// TwinCAT 3 PLC project Main_PLC
// ProgramVersion: 3.1.4024.0
// libraries:
//   Tc2_Math, * (Beckhoff Automation GmbH)
//   Tc2_Standard, * (Beckhoff Automation GmbH)
//   Tc2_System, * (Beckhoff Automation GmbH)
//   Tc3_Module, * (Beckhoff Automation GmbH)
// project tree:
//   DUTs/ E_Mode.TcDUT, ST_HmiControl.TcDUT, ST_AutoControlSwitch.TcDUT
//   GVLs/ gHMI.TcGVL, gIO.TcGVL
//   / PlcTask.TcTTO
//   POUs/Function Blocks/ FB_MockTank.TcPOU, FB_StopWatch.TcPOU, FB_SwitchSingleThrow.TcPOU, FB_TankControl.TcPOU
//   POUs/Function/Utilities/ F_Clear.TcPOU, F_Compare.TcPOU, F_Copy.TcPOU
//   POUs/ MAIN.TcPOU
// real-time tasks:
//   TASK PlcTask: cycle T#10ms, priority 20, ADS port 350
// I/O:
//   DEVICE EtherCAT Interface 1 (EK1100) (disabled), AmsNetId 10.186.0.125.2.1
//     Coupler 1 [EK1100 EtherCAT Coupler (2A E-Bus)]
//       Digital Input 1 (EL1008) [EL1008 8Ch. Dig. Input 24V, 3ms]
//       Digital Output 1 (EL2008) [EL2008 8Ch. Dig. Output 24V, 0.5A]
// variable links:
//   Main PLC/Main PLC Instance <-> EtherCAT Interface 1 (EK1100)/Coupler 1/Digital Input 1 (EL1008)
//     PlcTask Inputs/gIO.I[{0..7}] <-> Channel {1..8}/Input  (8 links)
//   Main PLC/Main PLC Instance <-> EtherCAT Interface 1 (EK1100)/Coupler 1/Digital Output 1 (EL2008)
//     PlcTask Outputs/gIO.Q[{0..7}] <-> Channel {1..8}/Output  (8 links)

CONFIGURATION Main_PLC
    RESOURCE PLC ON TwinCAT3
        TASK PlcTask(INTERVAL := T#10ms, PRIORITY := 20);
        PROGRAM MAIN WITH PlcTask : MAIN;
    END_RESOURCE
END_CONFIGURATION

// ---- DUTs/E_Mode.TcDUT
{attribute 'qualified_only'}
{attribute 'strict'}
TYPE E_Mode :
(
	Manual, Auto
)USINT;
END_TYPE

// ---- DUTs/ST_HmiControl.TcDUT
TYPE ST_HmiControl :
STRUCT
	Lamp: WORD;
	Button: WORD;
	Interlock: WORD;
END_STRUCT
END_TYPE

// ---- DUTs/ST_AutoControlSwitch.TcDUT
TYPE ST_AutoControlSwitch :
STRUCT
	bExecute: BOOL;
	bDone: BOOL;
	bError: BOOL;
END_STRUCT
END_TYPE

// ---- GVLs/gHMI.TcGVL
{attribute 'qualified_only'}
VAR_GLOBAL
END_VAR

// ---- GVLs/gIO.TcGVL
VAR_GLOBAL
	I AT %I*: ARRAY[0..7] OF BOOL;
	Q AT %Q*: ARRAY[0..7] OF BOOL;
END_VAR

// ---- POUs/MAIN.TcPOU
PROGRAM MAIN
VAR
	fbTankControl: FB_TankControl;
	fbMockTank: FB_MockTank;
	
	{attribute 'OPC.UA.DA' := '1'}
	stTankPumpCtrl: ST_HmiControl;
	
	{attribute 'OPC.UA.DA' := '1'}
	bHmiReset: BOOL;
	
	{attribute 'OPC.UA.DA' := '1'}
	eHmiMode: E_Mode;
	
	{attribute 'OPC.UA.DA':='1'}
	{attribute 'OPC.UA.DA.Access':='1'}
	rTankVolume: REAL;
	
	{attribute 'OPC.UA.DA':='1'}
	{attribute 'OPC.UA.DA.Access':='1'}
	rConsumptionRate: REAL;
	
	{attribute 'OPC.UA.DA':='1'}
	{attribute 'OPC.UA.DA.Access':='1'}
	nAlarmBits: DWORD;
	
	nLiveAlarmBits: DWORD;
END_VAR

fbMockTank(
	bEnable:= fbMockTank.bEnable, 
	bPumpOn:= Q[0], 
	rPumpFillRate:= fbMockTank.rPumpFillRate, 
	rCapacity:= fbMockTank.rCapacity, 
	tSamplingRate:= fbMockTank.tSamplingRate,
	nLowLevelSensorPos:= fbMockTank.nLowLevelSensorPos, 
	nHighLevelSensorPos:= fbMockTank.nHighLevelSensorPos, 
	rVolume=> rTankVolume, 
	rConsumption=> rConsumptionRate, 
	bLowLevel=>, 
	bHighLevel=> );

IF fbMockTank.bEnable THEN	
	I[0]:= fbMockTank.bLowLevel;
	I[1]:= fbMockTank.bHighLevel;
END_IF

fbTankControl(
	bEnableFillTimeout:= fbTankControl.bEnableFillTimeout, 
	eMode:= eHmiMode, 
	bReset:= fbTankControl.bReset, 
	tHighLevelSensorDly:= fbTankControl.tHighLevelSensorDly, 
	tLowLevelSensorDly:= fbTankControl.tLowLevelSensorDly, 
	tFillTimeout:= fbTankControl.tFillTimeout, 
	bPumpOnOutput:= Q[0], 
	bHighLevelSensor:= I[1], 
	bLowLevelSensor:= I[0], 
	stPumpHmiControl:= stTankPumpCtrl);
	
IF bHmiReset THEN
	F_Clear(nAlarmBits);
END_IF

nLiveAlarmBits.0:= NOT I[0];
nLiveAlarmBits.1:= I[1];

nAlarmBits:= nAlarmBits OR nLiveAlarmBits;

END_PROGRAM

// ---- POUs/Function Blocks/FB_TankControl.TcPOU
FUNCTION_BLOCK FB_TankControl
VAR_INPUT
	bEnableFillTimeout: BOOL;
	eMode: E_Mode;
	bReset: BOOL;
	tHighLevelSensorDly: TIME:= T#0.2S;
	tLowLevelSensorDly: TIME:= T#0.2S;
	tFillTimeout: TIME:= T#10S;
END_VAR
VAR_IN_OUT
	bPumpOnOutput: BOOL;
	bHighLevelSensor: BOOL;
	bLowLevelSensor: BOOL;
	stPumpHmiControl: ST_HmiControl;
END_VAR
VAR
	tonHighLevelSensorDly: TON;
	tonLowLevelSensorDly: TON;
	tonFillTimeout: TON;
	
	stPumpOnAuto: ST_AutoControlSwitch;
	fbPumpControl: FB_SwitchSingleThrow;
END_VAR

tonHighLevelSensorDly(IN:= bHighLevelSensor, PT:= tHighLevelSensorDly, Q=> , ET=> );
tonLowLevelSensorDly(IN:= NOT bLowLevelSensor, PT:= tLowLevelSensorDly, Q=> , ET=> );

tonFillTimeout(IN:= bEnableFillTimeout, PT:= tFillTimeout, Q=> , ET=> );

fbPumpControl(
	bManualMode:= eMode = E_Mode.Manual, 
	bReset:= bReset,  
	bSensor:= TRUE, 
	bInterlock:= tonHighLevelSensorDly.Q, 
	tTimeout:= , 
	tMinSensorOn:= , 
	stAuto:= stPumpOnAuto, 
	stHmiControl:= stPumpHmiControl,
	bError=> , 
	sErrorMsg=> , 
	bSwitch=> bPumpOnOutput, 
	bOverrideState=> );

IF eMode = E_Mode.Auto THEN
	stPumpOnAuto.bExecute:= 
		NOT (tonHighLevelSensorDly.Q OR tonFillTimeout.Q) AND (stPumpOnAuto.bExecute OR tonLowLevelSensorDly.Q);
END_IF

END_FUNCTION_BLOCK

// ---- POUs/Function Blocks/FB_SwitchSingleThrow.TcPOU
FUNCTION_BLOCK FB_SwitchSingleThrow
VAR_INPUT
	bManualMode: BOOL;
	bReset: BOOL;
	bSensor: BOOL;
	bInterlock: BOOL;
	tTimeout: TIME:= tDefaultTimeOut;
	tMinSensorOn: TIME:= tDefaultMinSensorOn;
END_VAR
VAR_IN_OUT
	stAuto: ST_AutoControlSwitch;
	stHmiControl: ST_HmiControl;
END_VAR
VAR_OUTPUT
	bError: BOOL;
	sErrorMsg: STRING(100);
	bSwitch: BOOL;
	
	bOverrideState: BOOL;
END_VAR
VAR
	tonPulse_Delay: Ton;
	tonSeqDelay: Ton;
	tonSeqTimeout: Ton;	
	
	rtReset: R_TRIG;
	
	nCurrentState: BYTE;
	nAutoState: BYTE;
	
	rtHome_Execute_HMI: R_TRIG;
	rtAction_Execute_HMI: R_TRIG;
	
	ton_DoneResetTimeout: TON;
	
	_bSwitch: BOOL;
END_VAR
VAR CONSTANT
	tDefaultMinPulseOn: TIME:= T#2S;
	tDefaultMinSensorOn: TIME:= T#0.1S;
	tDefaultTimeOut: TIME:= T#10S;
	tDefaultResetDone: TIME:= T#1S;
END_VAR

tonSeqDelay(
	IN:= bSensor,
	PT:= tMinSensorOn);
	
tonSeqTimeout(
	IN:= stAuto.bExecute AND NOT (stAuto.bDone OR stAuto.bError OR bManualMode),
	PT:= tTimeout);
	
ton_DoneResetTimeout(
	IN:= stAuto.bDone AND NOT bSensor,
	PT:= tDefaultResetDone);
	
IF ton_DoneResetTimeout.Q THEN
	F_Clear(stAuto.bDone);
END_IF
	
rtReset(CLK:= bReset);

bError:= stAuto.bError;

rtHome_Execute_HMI(CLK:= stHmiControl.Button.0);
rtAction_Execute_HMI(CLK:= stHmiControl.Button.1);

IF rtReset.Q AND bError THEN	
	stAuto.bError:= FALSE;
	sErrorMsg:= '';
END_IF

IF tonPulse_Delay.Q THEN
	F_Clear(stHmiControl);
	F_Clear(stAuto.bExecute);
	F_Clear(_bSwitch);
END_IF
IF bManualMode THEN
	IF rtHome_Execute_HMI.Q THEN
		stHmiControl.Button.1:= FALSE;
		_bSwitch:= FALSE;
	ELSIF rtAction_Execute_HMI.Q THEN
		IF bInterlock THEN
			stHmiControl.Button.1:= FALSE;
		ELSE
			stHmiControl.Button.0:= FALSE;
			_bSwitch:= TRUE;
		END_IF
	END_IF
	stAuto.bExecute:= stHmiControl.Button.1;
ELSE 
	IF NOT (bError AND stAuto.bExecute) THEN
		IF stAuto.bExecute THEN
			IF NOT bInterlock THEN
				_bSwitch:= TRUE;
			END_IF
		ELSE
			_bSwitch:= FALSE;
		END_IF
		IF tonSeqTimeout.Q THEN
			stAuto.bError:= TRUE;
			IF bInterlock THEN
				sErrorMsg:= 'Interlock Error';
			ELSE 
				sErrorMsg:= 'Timeout Error';
			END_IF
		END_IF
	END_IF
	stHmiControl.Button.1:= stAuto.bExecute;
	stHmiControl.Button.0:= NOT stAuto.bExecute;
END_IF

stHmiControl.Interlock.1:= bInterlock;
stAuto.bDone:= stAuto.bExecute AND (tonSeqDelay.Q OR stAuto.bDone) AND NOT stAuto.bError;

nCurrentState.0:= bSwitch;
IF NOT bManualMode THEN
	nAutoState:= nCurrentState;
END_IF
bOverrideState:= nCurrentState <> nAutoState;

bSwitch:= _bSwitch;

END_FUNCTION_BLOCK

// ---- POUs/Function/Utilities/F_Clear.TcPOU
FUNCTION F_Clear : BOOL //size of data type should not exceed double integer maximum value
VAR_INPUT
	Target: ANY;
END_VAR
VAR
END_VAR

MemSet(
	DestAddr       	:= Target.pValue, 
    FillByte    	:= 0, 
    n   			:= DINT_TO_UDINT(Target.diSize)
);

END_FUNCTION

// ---- POUs/Function Blocks/FB_MockTank.TcPOU
FUNCTION_BLOCK FB_MockTank
VAR_INPUT
	bEnable: BOOL;
	bPumpOn: BOOL;
	rPumpFillRate: REAL:= 50; //litres per second
	rCapacity: REAL:= 500; //litres
	nLowLevelSensorPos: REAL:= 0.2*rCapacity; //percent
	nHighLevelSensorPos: REAL:= 0.8*rCapacity; //percent
	tSamplingRate: TIME:= T#100MS;
END_VAR
VAR_OUTPUT
	rVolume: REAL;
	rConsumption: REAL;
	bLowLevel: BOOL;
	bHighLevel: BOOL;
END_VAR
VAR
	tonConsumptionPeriod: TON;
	rFillRate: REAL;
	fbRandom: DRAND;
	tonSamplingRate: TON;
	rFillRateFactor: REAL;
END_VAR

VAR CONSTANT
	
END_VAR

bLowLevel:= rVolume > nLowLevelSensorPos;
bHighLevel:= rVolume > nHighLevelSensorPos;

tonConsumptionPeriod(IN:= bEnable AND NOT tonConsumptionPeriod.Q, PT:= , Q=> , ET=> );
tonSamplingRate(IN:= bEnable AND NOT tonSamplingRate.Q, PT:= tSamplingRate, Q=> , ET=> );
IF bPumpOn THEN
	rFillRate:= rPumpFillRate;
ELSE
	rFillRate:= 0.0;
END_IF

IF bEnable THEN
	rFillRateFactor:= TIME_TO_REAL(tonSamplingRate.PT)/1000;
	IF tonConsumptionPeriod.Q THEN
		fbRandom(seed:=LREAL_TO_INT(fbRandom.Num));
		IF rConsumption = 0.0 THEN
			rConsumption:= fbRandom.Num*fbRandom.Num*20;
			tonConsumptionPeriod.PT:= LREAL_TO_TIME(fbRandom.Num*10000);
		ELSE
			rConsumption:= 0.0;
			tonConsumptionPeriod.PT:= LREAL_TO_TIME(fbRandom.Num*2000);
		END_IF
	END_IF
	IF rVolume < 0.1 THEN
		rConsumption:= 0.0;
	END_IF
	IF tonSamplingRate.Q THEN
		rVolume:= rVolume + (rFillRate - rConsumption)*rFillRateFactor;
	END_IF
END_IF

END_FUNCTION_BLOCK

// ---- POUs/Function Blocks/FB_StopWatch.TcPOU
FUNCTION_BLOCK FB_StopWatch
VAR_INPUT
	bStart: BOOL;
	bReset: BOOL;
END_VAR
VAR_IN_OUT
	tElapsedTime: TIME;
END_VAR
VAR
	tStartTime: TIME;
	rtReset: R_TRIG;
	tLastElapsedTime: TIME;
END_VAR

rtReset(CLK:= bReset);
IF rtReset.Q THEN
	F_Clear(tLastElapsedTime);
	F_Clear(tStartTime);
END_IF

IF bStart AND tStartTime = T#0MS THEN
	tStartTime:= TIME();
ELSIF NOT bStart AND tStartTime > T#0MS THEN
	tLastElapsedTime:= tLastElapsedTime + TIME() - tStartTime;
	F_Clear(tStartTime);
END_IF

IF tStartTime > T#0MS THEN
	tElapsedTime:= tLastElapsedTime + TIME() - tStartTime;
ELSIF tLastElapsedTime = T#0S AND tElapsedTime > T#0S THEN
	tLastElapsedTime:= tElapsedTime;
ELSE
	tElapsedTime:= tLastElapsedTime;
END_IF

END_FUNCTION_BLOCK

// ---- POUs/Function/Utilities/F_Compare.TcPOU
FUNCTION F_Compare : BOOL
VAR_INPUT
	Var1: ANY;
	Var2: ANY;
END_VAR
VAR
	nDiff: DINT:= -1; 
END_VAR

IF Var1.diSize = Var2.diSize THEN
	nDiff:= MEMCMP(
			pBuf1:= Var1.pValue, 
			pBuf2:= Var2.pValue, 
			n:= DINT_TO_UDINT(Var2.diSize));
END_IF

F_Compare:= nDiff = 0;

END_FUNCTION

// ---- POUs/Function/Utilities/F_Copy.TcPOU
FUNCTION F_Copy : BOOL //data should of child or parent
VAR_INPUT
	Target: ANY;
	Source: ANY;
END_VAR
VAR
	nSize: UDINT;
END_VAR

IF Target.diSize > Source.diSize THEN
	nSize:= DINT_TO_UDINT(Source.diSize);
ELSE
	nSize:= DINT_TO_UDINT(Target.diSize);
END_IF

MEMCPY(
	destAddr		:= Target.pValue,
	srcAddr			:= Source.pValue,
	n				:= nSize
);

END_FUNCTION
